// TwinCAT 3 PLC project Prototype_Pattern
// ProgramVersion: 3.1.4024.0
// libraries:
//   Tc2_Standard, * (Beckhoff Automation GmbH)
//   Tc2_System, * (Beckhoff Automation GmbH)
//   Tc3_Module, * (Beckhoff Automation GmbH)
// project tree:
//   Classes/ RecipeRunner.TcPOU
//   Interfaces/ ITF_Cloneable.TcIO, ITF_RecipePoint.TcIO
//   / PlcTask.TcTTO
//   POUs/ MAIN.TcPOU
//   Prototypes/ RecipePoint.TcPOU
// (motion and I/O tree: see PLC project simple_factory_pattern)
// real-time tasks:
//   TASK PlcTask: cycle T#10ms, priority 20, ADS port 350
//   TASK PlcTask1: cycle T#10ms, priority 21, ADS port 351
//   TASK PlcTask2: cycle T#10ms, priority 22, ADS port 352
//   TASK PlcTask3: cycle T#10ms, priority 23, ADS port 353
//   TASK PlcTask4: cycle T#10ms, priority 24, ADS port 354
//   TASK PlcTask5: cycle T#10ms, priority 25, ADS port 355
//   TASK PlcTask6: cycle T#10ms, priority 26, ADS port 356
//   TASK PlcTask7: cycle T#10ms, priority 27, ADS port 357
//   TASK PlcTask8: cycle T#10ms, priority 28, ADS port 358
//   TASK PlcTask9: cycle T#10ms, priority 29, ADS port 359
//   TASK PlcTask10: cycle T#10ms, priority 30, ADS port 360
//   TASK PlcTask11: cycle T#10ms, priority 31, ADS port 361

CONFIGURATION Prototype_Pattern
    RESOURCE PLC ON TwinCAT3
        TASK PlcTask(INTERVAL := T#10ms, PRIORITY := 31);
        PROGRAM MAIN WITH PlcTask : MAIN;
    END_RESOURCE
END_CONFIGURATION

// ---- Interfaces/ITF_Cloneable.TcIO
INTERFACE ITF_Cloneable

END_INTERFACE

// ---- Interfaces/ITF_RecipePoint.TcIO
INTERFACE ITF_RecipePoint

PROPERTY XPoint : LREAL
GET
END_GET
SET
END_SET
END_PROPERTY

PROPERTY YPoint : LREAL
GET
END_GET
SET
END_SET
END_PROPERTY

PROPERTY ZPoint : LREAL
GET
END_GET
SET
END_SET
END_PROPERTY

END_INTERFACE

// ---- POUs/MAIN.TcPOU
PROGRAM MAIN
VAR
	runner : RecipeRunner;
	recipePt : RecipePoint := (XPoint := 10.0, YPoint := 1.0, ZPoint := 2.0);
	CreatePoint: BOOL;
	newXPos : LREAL;
	runRecipe: BOOL;
END_VAR

IF CreatePoint THEN
	CreatePoint := FALSE;
	runner.AddRecipePoint(recipePt.Clone(xPoint := newXPos,yPoint := 0.0, zPoint := 0.0));
END_IF

IF runRecipe THEN
	IF runner.RunRecipe() THEN
		runRecipe := FALSE;
	END_IF
END_IF

runner.Cycle();

END_PROGRAM

// ---- Classes/RecipeRunner.TcPOU
FUNCTION_BLOCK RecipeRunner
VAR
	SetPoint : ARRAY[0..9] OF ITF_RecipePoint;
	NumberOfPoints : INT;
	BasePoint : RecipePoint := (XPoint := 19.0, YPoint := 23.0, ZPoint := 2.1);
	i: INT;
	TargetXPos : LREAL;
	recipeDelay : TON := (PT := t#2s);
END_VAR

METHOD AddRecipePoint : BOOL
VAR_INPUT
	point : ITF_RecipePoint;
END_VAR
IF point <> 0 AND NumberOfPoints < 10 THEN
	SetPoint[NumberOfPoints] := point;
	NumberOfPoints := NumberOfPoints + 1;
END_IF
END_METHOD

METHOD Cycle : BOOL
VAR_INPUT
END_VAR
recipeDelay();
END_METHOD

METHOD RunRecipe : BOOL
VAR_INPUT
END_VAR
IF i <= NumberOfPoints THEN
	IF SetPoint[i] <> 0 THEN
		TargetXPos := SetPoint[i].XPoint;
		recipeDelay.IN := TRUE;
		IF recipeDelay.Q THEN
			i := i + 1;
			recipeDelay.IN := FALSE;
		END_IF
	END_IF
ELSE
	RunRecipe := TRUE;
	i := 0;
END_IF
END_METHOD

END_FUNCTION_BLOCK

// ---- Prototypes/RecipePoint.TcPOU
{attribute 'enable_dynamic_creation'}
FUNCTION_BLOCK RecipePoint IMPLEMENTS ITF_Cloneable, ITF_RecipePoint
VAR
	_xPoint : LREAL;
	_yPoint : LREAL;
	_zPoint : lreal;
END_VAR

METHOD  Clone : ITF_RecipePoint
VAR_INPUT
	xPoint : LREAL;
	yPoint : LREAL;
	zPoint : LREAL;
END_VAR
VAR
	pFB : POINTER TO RecipePoint;
END_VAR
pFB := __NEW(RecipePoint);
Clone := pFB^;
IF xPoint = 0.0 THEN
	Clone.XPoint := _xPoint;
ELSE
	Clone.XPoint := xPoint;
END_IF
IF yPoint = 0.0 THEN
	Clone.YPoint := _yPoint;
ELSE
	Clone.YPoint := yPoint;
END_IF
IF zPoint = 0.0 THEN
	Clone.ZPoint := _zPoint;
ELSE
	Clone.ZPoint := zPoint;
END_IF
END_METHOD

PROPERTY XPoint : LREAL
GET
XPoint := _xPoint;
END_GET
SET
_xPoint := XPoint;
END_SET
END_PROPERTY

PROPERTY YPoint : LREAL
GET
YPoint := _yPoint;
END_GET
SET
_yPoint := YPoint;
END_SET
END_PROPERTY

PROPERTY ZPoint : LREAL
GET
ZPoint := _zPoint;
END_GET
SET
_zPoint := ZPoint;
END_SET
END_PROPERTY

END_FUNCTION_BLOCK
